FUNCTION_BLOCK FB_ErrorReset
VAR_INPUT
	bEnbale							: BOOL;
	bResetErrors					: BOOL;
END_VAR
VAR_OUTPUT
	bAllErrorsCleared				: BOOL;
END_VAR
VAR
	tonCaseDelay									: ARRAY[0..10] OF TON;
	rTrigCase										: ARRAY[0..10] OF R_TRIG;
END_VAR
VAR_IN_OUT
	stSmacIO						: ST_SMAC_I_O;
	bHomeError_L					: BOOL;
	bHomeError_R					: BOOL;
	bPhasingError_L					: BOOL;
	bPhasingError_R					: BOOL;
	bCycleError						: BOOL;
	
	
END_VAR

IF bEnbale THEN
	ACT_ErrorReset();
END_IF

ACTION ACT_ErrorReset:
IF bResetErrors THEN
	
	bHomeError_L							:= FALSE;				
	bHomeError_R							:= FALSE;
	bPhasingError_L							:= FALSE;
	bPhasingError_R							:= FALSE;
	bCycleError								:= FALSE;

stSmacIO.qnControlWordLinear				:= 5;

IF tonCaseDelay[0].Q THEN
	stSmacIO.qnControlWordRotative				:= 5;
END_IF


IF (bHomeError_L				= FALSE) AND 
	(bHomeError_R				= FALSE) AND
	(bPhasingError_L			= FALSE) AND
	(bPhasingError_R			= FALSE) AND
	(bCycleError				= FALSE) AND NOT
	stSmacIO.inStatusWordLinear.13		 AND NOT
	stSmacIO.inStatusWordRotative.13	 THEN
	bAllErrorsCleared			:= TRUE;
ELSE bAllErrorsCleared			:= FALSE;
END_IF
END_IF
END_ACTION

ACTION ACT_TimTrig:
//TIMERS
	tonCaseDelay[0](IN := stSmacIO.qnControlWordLinear	= 5, PT:= T#500MS);
END_ACTION

END_FUNCTION_BLOCK

(* stored: Version 1.1.0.1, ProductVersion 3.1.4024.12
   POU FB_ErrorReset: Id {6158f349-3279-41a3-9438-bb7194c818ec}, SpecialFunc None
   Action ACT_ErrorReset: Id {a262ee29-d167-466d-a381-4ddba3c5f31f}
   Action ACT_TimTrig: Id {93658345-a537-4237-a6f8-2a15bd6122e2} *)
